{attribute 'pack_mode' := '1'}
TYPE TMDE :
STRUCT
	dwPceBad		: DWORD;
	dwPceGood		: DWORD;
	iPertCode		: INT;
	iStatus			: INT;
END_STRUCT
END_TYPE

(* stored: Version 1.1.0.1, ProductVersion 3.1.4022.12
   DUT TMDE: Id {653d1d15-d9a8-46f4-8954-9c1bb17af9b8} *)
